   //    faSingleStepModeUnit22 : Bool;
   //    faSingleModeUnit22 : Bool;
   //    fctBit1ClampingUnit22 : Bool;
   //    fctBit2ClampingUnit22 : Bool;
   //    fctBit3ClampingUnit22 : Bool;
   //    prealarmOnUnit23 : Bool;
   //    messageOnUnit23 : Bool;
   //    faSetupModeUnit23 : Bool;
   //    faSingleStepModeUnit23 : Bool;
   //    faSingleModeUnit23 : Bool;
   //    fctBit1ClampingUnit23 : Bool;
   //    fctBit2ClampingUnit23 : Bool;
   //    fctBit3ClampingUnit23 : Bool;
   //    prealarmOnUnit24 : Bool;
   //    messageOnUnit24 : Bool;
   //    faSetupModeUnit24 : Bool;
   //    faSingleStepModeUnit24 : Bool;
   //    faSingleModeUnit24 : Bool;
   //    fctBit1ClampingUnit24 : Bool;
   //    fctBit2ClampingUnit24 : Bool;
   //    fctBit3ClampingUnit24 : Bool;
   //    prealarmOnUnit25 : Bool;
   //    messageOnUnit25 : Bool;
   //    faSetupModeUnit25 : Bool;
   //    faSingleStepModeUnit25 : Bool;
   //    faSingleModeUnit25 : Bool;
   //    fctBit1ClampingUnit25 : Bool;
   //    fctBit2ClampingUnit25 : Bool;
   //    fctBit3ClampingUnit25 : Bool;
   //    prealarmOnUnit26 : Bool;
   //    messageOnUnit26 : Bool;
   //    faSetupModeUnit26 : Bool;
   //    faSingleStepModeUnit26 : Bool;
   //    faSingleModeUnit26 : Bool;
   //    fctBit1ClampingUnit26 : Bool;
   //    fctBit2ClampingUnit26 : Bool;
   //    fctBit3ClampingUnit26 : Bool;
   //    prealarmOnUnit27 : Bool;
   //    messageOnUnit27 : Bool;
   //    faSetupModeUnit27 : Bool;
   //    faSingleStepModeUnit27 : Bool;
   //    faSingleModeUnit27 : Bool;
   //    fctBit1ClampingUnit27 : Bool;
   //    fctBit2ClampingUnit27 : Bool;
   //    fctBit3ClampingUnit27 : Bool;
   //    prealarmOnUnit28 : Bool;
   //    messageOnUnit28 : Bool;
   //    faSetupModeUnit28 : Bool;
   //    faSingleStepModeUnit28 : Bool;
   //    faSingleModeUnit28 : Bool;
   //    fctBit1ClampingUnit28 : Bool;
   //    fctBit2ClampingUnit28 : Bool;
   //    fctBit3ClampingUnit28 : Bool;
   //    prealarmOnUnit29 : Bool;
   //    messageOnUnit29 : Bool;
   //    faSetupModeUnit29 : Bool;
   //    faSingleStepModeUnit29 : Bool;
   //    faSingleModeUnit29 : Bool;
   //    fctBit1ClampingUnit29 : Bool;
   //    fctBit2ClampingUnit29 : Bool;
   //    fctBit3ClampingUnit29 : Bool;
   //    prealarmOnUnit30 : Bool;
   //    messageOnUnit30 : Bool;
   //    faSetupModeUnit30 : Bool;
   //    faSingleStepModeUnit30 : Bool;
   //    faSingleModeUnit30 : Bool;
   //    fctBit1ClampingUnit30 : Bool;
   //    fctBit2ClampingUnit30 : Bool;
   //    fctBit3ClampingUnit30 : Bool;
   //    prealarmOnUnit31 : Bool;
   //    messageOnUnit31 : Bool;
   //    faSetupModeUnit31 : Bool;
   //    faSingleStepModeUnit31 : Bool;
   //    faSingleModeUnit31 : Bool;
   //    fctBit1ClampingUnit31 : Bool;
   //    fctBit2ClampingUnit31 : Bool;
   //    fctBit3ClampingUnit31 : Bool;
   //    prealarmOnUnit32 : Bool;
   //    messageOnUnit32 : Bool;
   //    faSetupModeUnit32 : Bool;
   //    faSingleStepModeUnit32 : Bool;
   //    faSingleModeUnit32 : Bool;
   //    fctBit1ClampingUnit32 : Bool;
   //    fctBit2ClampingUnit32 : Bool;
   //    fctBit3ClampingUnit32 : Bool;
   //    prealarmOnUnit33 : Bool;
   //    messageOnUnit33 : Bool;
   //    faSetupModeUnit33 : Bool;
   //    faSingleStepModeUnit33 : Bool;
   //    faSingleModeUnit33 : Bool;
   //    fctBit1ClampingUnit33 : Bool;
   //    fctBit2ClampingUnit33 : Bool;
   //    fctBit3ClampingUnit33 : Bool;
   //    prealarmOnUnit34 : Bool;
   //    messageOnUnit34 : Bool;
   //    faSetupModeUnit34 : Bool;
   //    faSingleStepModeUnit34 : Bool;
   //    faSingleModeUnit34 : Bool;
   //    fctBit1ClampingUnit34 : Bool;
   //    fctBit2ClampingUnit34 : Bool;
   //    fctBit3ClampingUnit34 : Bool;
   //    prealarmOnUnit35 : Bool;
   //    messageOnUnit35 : Bool;
   //    faSetupModeUnit35 : Bool;
   //    faSingleStepModeUnit35 : Bool;
   //    faSingleModeUnit35 : Bool;
   //    fctBit1ClampingUnit35 : Bool;
   //    fctBit2ClampingUnit35 : Bool;
   //    fctBit3ClampingUnit35 : Bool;
   //    prealarmOnUnit36 : Bool;
   //    messageOnUnit36 : Bool;
   //    faSetupModeUnit36 : Bool;
   //    faSingleStepModeUnit36 : Bool;
   //    faSingleModeUnit36 : Bool;
   //    fctBit1ClampingUnit36 : Bool;
   //    fctBit2ClampingUnit36 : Bool;
   //    fctBit3ClampingUnit36 : Bool;
   //    prealarmOnUnit37 : Bool;
   //    messageOnUnit37 : Bool;
   //    faSetupModeUnit37 : Bool;
   //    faSingleStepModeUnit37 : Bool;
   //    faSingleModeUnit37 : Bool;
   //    fctBit1ClampingUnit37 : Bool;
   //    fctBit2ClampingUnit37 : Bool;
   //    fctBit3ClampingUnit37 : Bool;
   //    prealarmOnUnit38 : Bool;
   //    messageOnUnit38 : Bool;
   //    faSetupModeUnit38 : Bool;
   //    faSingleStepModeUnit38 : Bool;
   //    faSingleModeUnit38 : Bool;
   //    fctBit1ClampingUnit38 : Bool;
   //    fctBit2ClampingUnit38 : Bool;
   //    fctBit3ClampingUnit38 : Bool;
   //    prealarmOnUnit39 : Bool;
   //    messageOnUnit39 : Bool;
   //    faSetupModeUnit39 : Bool;
   //    faSingleStepModeUnit39 : Bool;
   //    faSingleModeUnit39 : Bool;
   //    fctBit1ClampingUnit39 : Bool;
   //    fctBit2ClampingUnit39 : Bool;
   //    fctBit3ClampingUnit39 : Bool;
   //    prealarmOnUnit40 : Bool;
   //    messageOnUnit40 : Bool;
   //    faSetupModeUnit40 : Bool;
   //    faSingleStepModeUnit40 : Bool;
   //    faSingleModeUnit40 : Bool;
   //    fctBit1ClampingUnit40 : Bool;
   //    fctBit2ClampingUnit40 : Bool;
   //    fctBit3ClampingUnit40 : Bool;
   //    targetCycleTimeCompleteMach : Word;
   //    targetCycleTime : Array[1..40] of Word;
   //    station : Array[1..40] of Word;
   //    directKeyScreen : Struct
   //       activeLine : Byte;
   //       singleMovementActive : Bool;
   //       singleLineSelected : Bool;
   //       singleLineRequestForLock : Bool;
   //       singleLineIsLockedByHMI : Bool;
   //       reserved2003p4 : Bool;
   //       reserved2003p5 : Bool;
   //       leftKeyPressedVDCK : Bool;
   //       rightKeyPressedVDCK : Bool;
   //    END_STRUCT;
   //    FC57_1 : DWord;
   //    FC57_2 : DWord;
   //    FC57_3 : Byte;
   //    FC57_4 : Byte;
   //    FC57_5 : Word;
   //    FC57_6 : Word;
   //    opKey2LeftVertical : Bool;
   //    opKey2RightVertical : Bool;
   //    opKey3LeftVertical : Bool;
   //    opKey3RightVertical : Bool;
   //    opKey4LeftVertical : Bool;
   //    opKey4RightVertical : Bool;
   //    opKey5LeftVertical : Bool;
   //    opKey5RightVertical : Bool;
   //    opKey6LeftVertical : Bool;
   //    opKey6RightVertical : Bool;
   //    opKey7LeftVertical : Bool;
   //    opKey7RightVertical : Bool;
   //    executionPlus : Bool;
   //    executionMinus : Bool;
   //    enableMotion : Bool;
   //    enablePCU : Bool;
   //    mppPlusKey : Bool;
   //    mppMinusKey : Bool;
   //    res2921 : Byte;
   //    typePreselectWorkpieceCode : Array[1..32] of Word;
   //    typePreselectColorChange : Array[1..32] of Bool;
   //    res2990 : Array[2990..2999] of Byte;
   //    unit1WorkpieceAMeas2 : Bool;
   //    unit1WorkpieceAMeas1 : Bool;
   //    unit1WorkpieceBMeas2 : Bool;
   //    unit1WorkpieceBMeas1 : Bool;
   //    unit1WorkpieceCMeas2 : Bool;
   //    unit1WorkpieceCMeas1 : Bool;
   //    unit1WorkpieceDMeas2 : Bool;
   //    unit1WorkpieceDMeas1 : Bool;
   //    unit1WorkpieceEMeas2 : Bool;
   //    unit1WorkpieceEMeas1 : Bool;
   //    unit1WorkpieceFMeas2 : Bool;
   //    unit1WorkpieceFMeas1 : Bool;
   //    unit1WorkpieceGMeas2 : Bool;
   //    unit1WorkpieceGMeas1 : Bool;
   //    unit1WorkpieceHMeas2 : Bool;
   //    unit1WorkpieceHMeas1 : Bool;
   //    unit2WorkpieceAMeas2 : Bool;
   //    unit2WorkpieceAMeas1 : Bool;
   //    unit2WorkpieceBMeas2 : Bool;
   //    unit2WorkpieceBMeas1 : Bool;
   //    unit2WorkpieceCMeas2 : Bool;
   //    unit2WorkpieceCMeas1 : Bool;
   //    unit2WorkpieceDMeas2 : Bool;
   //    unit2WorkpieceDMeas1 : Bool;
   //    unit2WorkpieceEMeas2 : Bool;
   //    unit2WorkpieceEMeas1 : Bool;
   //    unit2WorkpieceFMeas2 : Bool;
   //    unit2WorkpieceFMeas1 : Bool;
   //    unit2WorkpieceGMeas2 : Bool;
   //    unit2WorkpieceGMeas1 : Bool;
   //    unit2WorkpieceHMeas2 : Bool;
   //    unit2WorkpieceHMeas1 : Bool;
   //    unit3WorkpieceAMeas2 : Bool;
   //    unit3WorkpieceAMeas1 : Bool;
   //    unit3WorkpieceBMeas2 : Bool;
   //    unit3WorkpieceBMeas1 : Bool;
   //    unit3WorkpieceCMeas2 : Bool;
   //    unit3WorkpieceCMeas1 : Bool;
   //    unit3WorkpieceDMeas2 : Bool;
   //    unit3WorkpieceDMeas1 : Bool;
   //    unit3WorkpieceEMeas2 : Bool;
   //    unit3WorkpieceEMeas1 : Bool;
   //    unit3WorkpieceFMeas2 : Bool;
   //    unit3WorkpieceFMeas1 : Bool;
   //    unit3WorkpieceGMeas2 : Bool;
   //    unit3WorkpieceGMeas1 : Bool;
   //    unit3WorkpieceHMeas2 : Bool;
   //    unit3WorkpieceHMeas1 : Bool;
   //    unit4WorkpieceAMeas2 : Bool;
   //    unit4WorkpieceAMeas1 : Bool;
   //    unit4WorkpieceBMeas2 : Bool;
   //    unit4WorkpieceBMeas1 : Bool;
   //    unit4WorkpieceCMeas2 : Bool;
   //    unit4WorkpieceCMeas1 : Bool;
   //    unit4WorkpieceDMeas2 : Bool;
   //    unit4WorkpieceDMeas1 : Bool;
   //    unit4WorkpieceEMeas2 : Bool;
   //    unit4WorkpieceEMeas1 : Bool;
   //    unit4WorkpieceFMeas2 : Bool;
   //    unit4WorkpieceFMeas1 : Bool;
   //    unit4WorkpieceGMeas2 : Bool;
   //    unit4WorkpieceGMeas1 : Bool;
   //    unit4WorkpieceHMeas2 : Bool;
   //    unit4WorkpieceHMeas1 : Bool;
   //    unit5WorkpieceAMeas2 : Bool;
   //    unit5WorkpieceAMeas1 : Bool;
   //    unit5WorkpieceBMeas2 : Bool;
   //    unit5WorkpieceBMeas1 : Bool;
   //    unit5WorkpieceCMeas2 : Bool;
   //    unit5WorkpieceCMeas1 : Bool;
   //    unit5WorkpieceDMeas2 : Bool;
   //    unit5WorkpieceDMeas1 : Bool;
   //    unit5WorkpieceEMeas2 : Bool;
   //    unit5WorkpieceEMeas1 : Bool;
   //    unit5WorkpieceFMeas2 : Bool;
   //    unit5WorkpieceFMeas1 : Bool;
   //    unit5WorkpieceGMeas2 : Bool;
   //    unit5WorkpieceGMeas1 : Bool;
   //    unit5WorkpieceHMeas2 : Bool;
   //    unit5WorkpieceHMeas1 : Bool;
   //    unit6WorkpieceAMeas2 : Bool;
   //    unit6WorkpieceAMeas1 : Bool;
   //    unit6WorkpieceBMeas2 : Bool;
   //    unit6WorkpieceBMeas1 : Bool;
   //    unit6WorkpieceCMeas2 : Bool;
   //    unit6WorkpieceCMeas1 : Bool;
   //    unit6WorkpieceDMeas2 : Bool;
   //    unit6WorkpieceDMeas1 : Bool;
   //    unit6WorkpieceEMeas2 : Bool;
   //    unit6WorkpieceEMeas1 : Bool;
   //    unit6WorkpieceFMeas2 : Bool;
   //    unit6WorkpieceFMeas1 : Bool;
   //    unit6WorkpieceGMeas2 : Bool;
   //    unit6WorkpieceGMeas1 : Bool;
   //    unit6WorkpieceHMeas2 : Bool;
   //    unit6WorkpieceHMeas1 : Bool;
   //    unit7WorkpieceAMeas2 : Bool;
   //    unit7WorkpieceAMeas1 : Bool;
   //    unit7WorkpieceBMeas2 : Bool;
   //    unit7WorkpieceBMeas1 : Bool;
   //    unit7WorkpieceCMeas2 : Bool;
   //    unit7WorkpieceCMeas1 : Bool;
   //    unit7WorkpieceDMeas2 : Bool;
   //    unit7WorkpieceDMeas1 : Bool;
   //    unit7WorkpieceEMeas2 : Bool;
   //    unit7WorkpieceEMeas1 : Bool;
   //    unit7WorkpieceFMeas2 : Bool;
   //    unit7WorkpieceFMeas1 : Bool;
   //    unit7WorkpieceGMeas2 : Bool;
   //    unit7WorkpieceGMeas1 : Bool;
   //    unit7WorkpieceHMeas2 : Bool;
   //    unit7WorkpieceHMeas1 : Bool;
   //    unit8WorkpieceAMeas2 : Bool;
   //    unit8WorkpieceAMeas1 : Bool;
   //    unit8WorkpieceBMeas2 : Bool;
   //    unit8WorkpieceBMeas1 : Bool;
   //    unit8WorkpieceCMeas2 : Bool;
   //    unit8WorkpieceCMeas1 : Bool;
   //    unit8WorkpieceDMeas2 : Bool;
   //    unit8WorkpieceDMeas1 : Bool;
   //    unit8WorkpieceEMeas2 : Bool;
   //    unit8WorkpieceEMeas1 : Bool;
   //    unit8WorkpieceFMeas2 : Bool;
   //    unit8WorkpieceFMeas1 : Bool;
   //    unit8WorkpieceGMeas2 : Bool;
   //    unit8WorkpieceGMeas1 : Bool;
   //    unit8WorkpieceHMeas2 : Bool;
   //    unit8WorkpieceHMeas1 : Bool;
   //    unit9WorkpieceAMeas2 : Bool;
   //    unit9WorkpieceAMeas1 : Bool;
   //    unit9WorkpieceBMeas2 : Bool;
   //    unit9WorkpieceBMeas1 : Bool;
   //    unit9WorkpieceCMeas2 : Bool;
   //    unit9WorkpieceCMeas1 : Bool;
   //    unit9WorkpieceDMeas2 : Bool;
   //    unit9WorkpieceDMeas1 : Bool;
   //    unit9WorkpieceEMeas2 : Bool;
   //    unit9WorkpieceEMeas1 : Bool;
   //    unit9WorkpieceFMeas2 : Bool;
   //    unit9WorkpieceFMeas1 : Bool;
   //    unit9WorkpieceGMeas2 : Bool;
   //    unit9WorkpieceGMeas1 : Bool;
   //    unit9WorkpieceHMeas2 : Bool;
   //    unit9WorkpieceHMeas1 : Bool;
   //    unit10WorkpieceAMeas2 : Bool;
   //    unit10WorkpieceAMeas1 : Bool;
   //    unit10WorkpieceBMeas2 : Bool;
   //    unit10WorkpieceBMeas1 : Bool;
   //    unit10WorkpieceCMeas2 : Bool;
   //    unit10WorkpieceCMeas1 : Bool;
   //    unit10WorkpieceDMeas2 : Bool;
   //    unit10WorkpieceDMeas1 : Bool;
   //    unit10WorkpieceEMeas2 : Bool;
   //    unit10WorkpieceEMeas1 : Bool;
   //    unit10WorkpieceFMeas2 : Bool;
   //    unit10WorkpieceFMeas1 : Bool;
   //    unit10WorkpieceGMeas2 : Bool;
   //    unit10WorkpieceGMeas1 : Bool;
   //    unit10WorkpieceHMeas2 : Bool;
   //    unit10WorkpieceHMeas1 : Bool;
   //    unit11WorkpieceAMeas2 : Bool;
   //    unit11WorkpieceAMeas1 : Bool;
   //    unit11WorkpieceBMeas2 : Bool;
   //    unit11WorkpieceBMeas1 : Bool;
   //    unit11WorkpieceCMeas2 : Bool;
   //    unit11WorkpieceCMeas1 : Bool;
   //    unit11WorkpieceDMeas2 : Bool;
   //    unit11WorkpieceDMeas1 : Bool;
   //    unit11WorkpieceEMeas2 : Bool;
   //    unit11WorkpieceEMeas1 : Bool;
   //    unit11WorkpieceFMeas2 : Bool;
   //    unit11WorkpieceFMeas1 : Bool;
   //    unit11WorkpieceGMeas2 : Bool;
   //    unit11WorkpieceGMeas1 : Bool;
   //    unit11WorkpieceHMeas2 : Bool;
   //    unit11WorkpieceHMeas1 : Bool;
   //    unit12WorkpieceAMeas2 : Bool;
   //    unit12WorkpieceAMeas1 : Bool;
   //    unit12WorkpieceBMeas2 : Bool;
   //    unit12WorkpieceBMeas1 : Bool;
   //    unit12WorkpieceCMeas2 : Bool;
   //    unit12WorkpieceCMeas1 : Bool;
   //    unit12WorkpieceDMeas2 : Bool;
   //    unit12WorkpieceDMeas1 : Bool;
   //    unit12WorkpieceEMeas2 : Bool;
   //    unit12WorkpieceEMeas1 : Bool;
   //    unit12WorkpieceFMeas2 : Bool;
   //    unit12WorkpieceFMeas1 : Bool;
   //    unit12WorkpieceGMeas2 : Bool;
   //    unit12WorkpieceGMeas1 : Bool;
   //    unit12WorkpieceHMeas2 : Bool;
   //    unit12WorkpieceHMeas1 : Bool;
   //    unit13WorkpieceAMeas2 : Bool;
   //    unit13WorkpieceAMeas1 : Bool;
   //    unit13WorkpieceBMeas2 : Bool;
   //    unit13WorkpieceBMeas1 : Bool;
   //    unit13WorkpieceCMeas2 : Bool;
   //    unit13WorkpieceCMeas1 : Bool;
   //    unit13WorkpieceDMeas2 : Bool;
   //    unit13WorkpieceDMeas1 : Bool;
   //    unit13WorkpieceEMeas2 : Bool;
   //    unit13WorkpieceEMeas1 : Bool;
   //    unit13WorkpieceFMeas2 : Bool;
   //    unit13WorkpieceFMeas1 : Bool;
   //    unit13WorkpieceGMeas2 : Bool;
   //    unit13WorkpieceGMeas1 : Bool;
   //    unit13WorkpieceHMeas2 : Bool;
   //    unit13WorkpieceHMeas1 : Bool;
   //    unit14WorkpieceAMeas2 : Bool;
   //    unit14WorkpieceAMeas1 : Bool;
   //    unit14WorkpieceBMeas2 : Bool;
   //    unit14WorkpieceBMeas1 : Bool;
   //    unit14WorkpieceCMeas2 : Bool;
   //    unit14WorkpieceCMeas1 : Bool;
   //    unit14WorkpieceDMeas2 : Bool;
   //    unit14WorkpieceDMeas1 : Bool;
   //    unit14WorkpieceEMeas2 : Bool;
   //    unit14WorkpieceEMeas1 : Bool;
   //    unit14WorkpieceFMeas2 : Bool;
   //    unit14WorkpieceFMeas1 : Bool;
   //    unit14WorkpieceGMeas2 : Bool;
   //    unit14WorkpieceGMeas1 : Bool;
   //    unit14WorkpieceHMeas2 : Bool;
   //    unit14WorkpieceHMeas1 : Bool;
   //    unit15WorkpieceAMeas2 : Bool;
   //    unit15WorkpieceAMeas1 : Bool;
   //    unit15WorkpieceBMeas2 : Bool;
   //    unit15WorkpieceBMeas1 : Bool;
   //    unit15WorkpieceCMeas2 : Bool;
   //    unit15WorkpieceCMeas1 : Bool;
   //    unit15WorkpieceDMeas2 : Bool;
   //    unit15WorkpieceDMeas1 : Bool;
   //    unit15WorkpieceEMeas2 : Bool;
   //    unit15WorkpieceEMeas1 : Bool;
   //    unit15WorkpieceFMeas2 : Bool;
   //    unit15WorkpieceFMeas1 : Bool;
   //    unit15WorkpieceGMeas2 : Bool;
   //    unit15WorkpieceGMeas1 : Bool;
   //    unit15WorkpieceHMeas2 : Bool;
   //    unit15WorkpieceHMeas1 : Bool;
   //    unit16WorkpieceAMeas2 : Bool;
   //    unit16WorkpieceAMeas1 : Bool;
   //    unit16WorkpieceBMeas2 : Bool;
   //    unit16WorkpieceBMeas1 : Bool;
   //    unit16WorkpieceCMeas2 : Bool;
   //    unit16WorkpieceCMeas1 : Bool;
   //    unit16WorkpieceDMeas2 : Bool;
   //    unit16WorkpieceDMeas1 : Bool;
   //    unit16WorkpieceEMeas2 : Bool;
   //    unit16WorkpieceEMeas1 : Bool;
   //    unit16WorkpieceFMeas2 : Bool;
   //    unit16WorkpieceFMeas1 : Bool;
   //    unit16WorkpieceGMeas2 : Bool;
   //    unit16WorkpieceGMeas1 : Bool;
   //    unit16WorkpieceHMeas2 : Bool;
   //    unit16WorkpieceHMeas1 : Bool;
   //    unit17WorkpieceAMeas2 : Bool;
   //    unit17WorkpieceAMeas1 : Bool;
   //    unit17WorkpieceBMeas2 : Bool;
   //    unit17WorkpieceBMeas1 : Bool;
   //    unit17WorkpieceCMeas2 : Bool;
   //    unit17WorkpieceCMeas1 : Bool;
   //    unit17WorkpieceDMeas2 : Bool;
   //    unit17WorkpieceDMeas1 : Bool;
   //    unit17WorkpieceEMeas2 : Bool;
   //    unit17WorkpieceEMeas1 : Bool;
   //    unit17WorkpieceFMeas2 : Bool;
   //    unit17WorkpieceFMeas1 : Bool;
   //    unit17WorkpieceGMeas2 : Bool;
   //    unit17WorkpieceGMeas1 : Bool;
   //    unit17WorkpieceHMeas2 : Bool;
   //    unit17WorkpieceHMeas1 : Bool;
   //    unit18WorkpieceAMeas2 : Bool;
   //    unit18WorkpieceAMeas1 : Bool;
   //    unit18WorkpieceBMeas2 : Bool;
   //    unit18WorkpieceBMeas1 : Bool;
   //    unit18WorkpieceCMeas2 : Bool;
   //    unit18WorkpieceCMeas1 : Bool;
   //    unit18WorkpieceDMeas2 : Bool;
   //    unit18WorkpieceDMeas1 : Bool;
   //    unit18WorkpieceEMeas2 : Bool;
   //    unit18WorkpieceEMeas1 : Bool;
   //    unit18WorkpieceFMeas2 : Bool;
   //    unit18WorkpieceFMeas1 : Bool;
   //    unit18WorkpieceGMeas2 : Bool;
   //    unit18WorkpieceGMeas1 : Bool;
   //    unit18WorkpieceHMeas2 : Bool;
   //    unit18WorkpieceHMeas1 : Bool;
   //    unit19WorkpieceAMeas2 : Bool;
   //    unit19WorkpieceAMeas1 : Bool;
   //    unit19WorkpieceBMeas2 : Bool;
   //    unit19WorkpieceBMeas1 : Bool;
   //    unit19WorkpieceCMeas2 : Bool;
   //    unit19WorkpieceCMeas1 : Bool;
   //    unit19WorkpieceDMeas2 : Bool;
   //    unit19WorkpieceDMeas1 : Bool;
   //    unit19WorkpieceEMeas2 : Bool;
   //    unit19WorkpieceEMeas1 : Bool;
   //    unit19WorkpieceFMeas2 : Bool;
   //    unit19WorkpieceFMeas1 : Bool;
   //    unit19WorkpieceGMeas2 : Bool;
   //    unit19WorkpieceGMeas1 : Bool;
   //    unit19WorkpieceHMeas2 : Bool;
   //    unit19WorkpieceHMeas1 : Bool;
   //    unit20WorkpieceAMeas2 : Bool;
   //    unit20WorkpieceAMeas1 : Bool;
   //    unit20WorkpieceBMeas2 : Bool;
   //    unit20WorkpieceBMeas1 : Bool;
   //    unit20WorkpieceCMeas2 : Bool;
   //    unit20WorkpieceCMeas1 : Bool;
   //    unit20WorkpieceDMeas2 : Bool;
   //    unit20WorkpieceDMeas1 : Bool;
   //    unit20WorkpieceEMeas2 : Bool;
   //    unit20WorkpieceEMeas1 : Bool;
   //    unit20WorkpieceFMeas2 : Bool;
   //    unit20WorkpieceFMeas1 : Bool;
   //    unit20WorkpieceGMeas2 : Bool;
   //    unit20WorkpieceGMeas1 : Bool;
   //    unit20WorkpieceHMeas2 : Bool;
   //    unit20WorkpieceHMeas1 : Bool;
   //    unit21WorkpieceAMeas2 : Bool;
   //    unit21WorkpieceAMeas1 : Bool;
   //    unit21WorkpieceBMeas2 : Bool;
   //    unit21WorkpieceBMeas1 : Bool;
   //    unit21WorkpieceCMeas2 : Bool;
   //    unit21WorkpieceCMeas1 : Bool;
   //    unit21WorkpieceDMeas2 : Bool;
   //    unit21WorkpieceDMeas1 : Bool;
   //    unit21WorkpieceEMeas2 : Bool;
   //    unit21WorkpieceEMeas1 : Bool;
   //    unit21WorkpieceFMeas2 : Bool;
   //    unit21WorkpieceFMeas1 : Bool;
   //    unit21WorkpieceGMeas2 : Bool;
   //    unit21WorkpieceGMeas1 : Bool;
   //    unit21WorkpieceHMeas2 : Bool;
   //    unit21WorkpieceHMeas1 : Bool;
   //    unit22WorkpieceAMeas2 : Bool;
   //    unit22WorkpieceAMeas1 : Bool;
   //    unit22WorkpieceBMeas2 : Bool;
   //    unit22WorkpieceBMeas1 : Bool;
   //    unit22WorkpieceCMeas2 : Bool;
   //    unit22WorkpieceCMeas1 : Bool;
   //    unit22WorkpieceDMeas2 : Bool;
   //    unit22WorkpieceDMeas1 : Bool;
   //    unit22WorkpieceEMeas2 : Bool;
   //    unit22WorkpieceEMeas1 : Bool;
   //    unit22WorkpieceFMeas2 : Bool;
   //    unit22WorkpieceFMeas1 : Bool;
   //    unit22WorkpieceGMeas2 : Bool;
   //    unit22WorkpieceGMeas1 : Bool;
   //    unit22WorkpieceHMeas2 : Bool;
   //    unit22WorkpieceHMeas1 : Bool;
   //    unit23WorkpieceAMeas2 : Bool;
   //    unit23WorkpieceAMeas1 : Bool;
   //    unit23WorkpieceBMeas2 : Bool;
   //    unit23WorkpieceBMeas1 : Bool;
   //    unit23WorkpieceCMeas2 : Bool;
   //    unit23WorkpieceCMeas1 : Bool;
   //    unit23WorkpieceDMeas2 : Bool;
   //    unit23WorkpieceDMeas1 : Bool;
   //    unit23WorkpieceEMeas2 : Bool;
   //    unit23WorkpieceEMeas1 : Bool;
   //    unit23WorkpieceFMeas2 : Bool;
   //    unit23WorkpieceFMeas1 : Bool;
   //    unit23WorkpieceGMeas2 : Bool;
   //    unit23WorkpieceGMeas1 : Bool;
   //    unit23WorkpieceHMeas2 : Bool;
   //    unit23WorkpieceHMeas1 : Bool;
   //    unit24WorkpieceAMeas2 : Bool;
   //    unit24WorkpieceAMeas1 : Bool;
   //    unit24WorkpieceBMeas2 : Bool;
   //    unit24WorkpieceBMeas1 : Bool;
   //    unit24WorkpieceCMeas2 : Bool;
   //    unit24WorkpieceCMeas1 : Bool;
   //    unit24WorkpieceDMeas2 : Bool;
   //    unit24WorkpieceDMeas1 : Bool;
   //    unit24WorkpieceEMeas2 : Bool;
   //    unit24WorkpieceEMeas1 : Bool;
   //    unit24WorkpieceFMeas2 : Bool;
   //    unit24WorkpieceFMeas1 : Bool;
   //    unit24WorkpieceGMeas2 : Bool;
   //    unit24WorkpieceGMeas1 : Bool;
   //    unit24WorkpieceHMeas2 : Bool;
   //    unit24WorkpieceHMeas1 : Bool;
   //    unit25WorkpieceAMeas2 : Bool;
   //    unit25WorkpieceAMeas1 : Bool;
   //    unit25WorkpieceBMeas2 : Bool;
   //    unit25WorkpieceBMeas1 : Bool;
   //    unit25WorkpieceCMeas2 : Bool;
   //    unit25WorkpieceCMeas1 : Bool;
   //    unit25WorkpieceDMeas2 : Bool;
   //    unit25WorkpieceDMeas1 : Bool;
   //    unit25WorkpieceEMeas2 : Bool;
   //    unit25WorkpieceEMeas1 : Bool;
   //    unit25WorkpieceFMeas2 : Bool;
   //    unit25WorkpieceFMeas1 : Bool;
   //    unit25WorkpieceGMeas2 : Bool;
   //    unit25WorkpieceGMeas1 : Bool;
   //    unit25WorkpieceHMeas2 : Bool;
   //    unit25WorkpieceHMeas1 : Bool;
   //    unit26WorkpieceAMeas2 : Bool;
   //    unit26WorkpieceAMeas1 : Bool;
   //    unit26WorkpieceBMeas2 : Bool;
   //    unit26WorkpieceBMeas1 : Bool;
   //    unit26WorkpieceCMeas2 : Bool;
   //    unit26WorkpieceCMeas1 : Bool;
   //    unit26WorkpieceDMeas2 : Bool;
   //    unit26WorkpieceDMeas1 : Bool;
   //    unit26WorkpieceEMeas2 : Bool;
   //    unit26WorkpieceEMeas1 : Bool;
   //    unit26WorkpieceFMeas2 : Bool;
   //    unit26WorkpieceFMeas1 : Bool;
   //    unit26WorkpieceGMeas2 : Bool;
   //    unit26WorkpieceGMeas1 : Bool;
   //    unit26WorkpieceHMeas2 : Bool;
   //    unit26WorkpieceHMeas1 : Bool;
   //    unit27WorkpieceAMeas2 : Bool;
   //    unit27WorkpieceAMeas1 : Bool;
   //    unit27WorkpieceBMeas2 : Bool;
   //    unit27WorkpieceBMeas1 : Bool;
   //    unit27WorkpieceCMeas2 : Bool;
   //    unit27WorkpieceCMeas1 : Bool;
   //    unit27WorkpieceDMeas2 : Bool;
   //    unit27WorkpieceDMeas1 : Bool;
   //    unit27WorkpieceEMeas2 : Bool;
   //    unit27WorkpieceEMeas1 : Bool;
   //    unit27WorkpieceFMeas2 : Bool;
   //    unit27WorkpieceFMeas1 : Bool;
   //    unit27WorkpieceGMeas2 : Bool;
   //    unit27WorkpieceGMeas1 : Bool;
   //    unit27WorkpieceHMeas2 : Bool;
   //    unit27WorkpieceHMeas1 : Bool;
   //    unit28WorkpieceAMeas2 : Bool;
   //    unit28WorkpieceAMeas1 : Bool;
   //    unit28WorkpieceBMeas2 : Bool;
   //    unit28WorkpieceBMeas1 : Bool;
   //    unit28WorkpieceCMeas2 : Bool;
   //    unit28WorkpieceCMeas1 : Bool;
   //    unit28WorkpieceDMeas2 : Bool;
   //    unit28WorkpieceDMeas1 : Bool;
   //    unit28WorkpieceEMeas2 : Bool;
   //    unit28WorkpieceEMeas1 : Bool;
   //    unit28WorkpieceFMeas2 : Bool;
   //    unit28WorkpieceFMeas1 : Bool;
   //    unit28WorkpieceGMeas2 : Bool;
   //    unit28WorkpieceGMeas1 : Bool;
   //    unit28WorkpieceHMeas2 : Bool;
   //    unit28WorkpieceHMeas1 : Bool;
   //    unit29WorkpieceAMeas2 : Bool;
   //    unit29WorkpieceAMeas1 : Bool;
   //    unit29WorkpieceBMeas2 : Bool;
   //    unit29WorkpieceBMeas1 : Bool;
   //    unit29WorkpieceCMeas2 : Bool;
   //    unit29WorkpieceCMeas1 : Bool;
   //    unit29WorkpieceDMeas2 : Bool;
   //    unit29WorkpieceDMeas1 : Bool;
   //    unit29WorkpieceEMeas2 : Bool;
   //    unit29WorkpieceEMeas1 : Bool;
   //    unit29WorkpieceFMeas2 : Bool;
   //    unit29WorkpieceFMeas1 : Bool;
   //    unit29WorkpieceGMeas2 : Bool;
   //    unit29WorkpieceGMeas1 : Bool;
   //    unit29WorkpieceHMeas2 : Bool;
   //    unit29WorkpieceHMeas1 : Bool;
   //    unit30WorkpieceAMeas2 : Bool;
   //    unit30WorkpieceAMeas1 : Bool;
   //    unit30WorkpieceBMeas2 : Bool;
   //    unit30WorkpieceBMeas1 : Bool;
   //    unit30WorkpieceCMeas2 : Bool;
   //    unit30WorkpieceCMeas1 : Bool;
   //    unit30WorkpieceDMeas2 : Bool;
   //    unit30WorkpieceDMeas1 : Bool;
   //    unit30WorkpieceEMeas2 : Bool;
   //    unit30WorkpieceEMeas1 : Bool;
   //    unit30WorkpieceFMeas2 : Bool;
   //    unit30WorkpieceFMeas1 : Bool;
   //    unit30WorkpieceGMeas2 : Bool;
   //    unit30WorkpieceGMeas1 : Bool;
   //    unit30WorkpieceHMeas2 : Bool;
   //    unit30WorkpieceHMeas1 : Bool;
   //    unit31WorkpieceAMeas2 : Bool;
   //    unit31WorkpieceAMeas1 : Bool;
   //    unit31WorkpieceBMeas2 : Bool;
   //    unit31WorkpieceBMeas1 : Bool;
   //    unit31WorkpieceCMeas2 : Bool;
   //    unit31WorkpieceCMeas1 : Bool;
   //    unit31WorkpieceDMeas2 : Bool;
   //    unit31WorkpieceDMeas1 : Bool;
   //    unit31WorkpieceEMeas2 : Bool;
   //    unit31WorkpieceEMeas1 : Bool;
   //    unit31WorkpieceFMeas2 : Bool;
   //    unit31WorkpieceFMeas1 : Bool;
   //    unit31WorkpieceGMeas2 : Bool;
   //    unit31WorkpieceGMeas1 : Bool;
   //    unit31WorkpieceHMeas2 : Bool;
   //    unit31WorkpieceHMeas1 : Bool;
   //    unit32WorkpieceAMeas2 : Bool;
   //    unit32WorkpieceAMeas1 : Bool;
   //    unit32WorkpieceBMeas2 : Bool;
   //    unit32WorkpieceBMeas1 : Bool;
   //    unit32WorkpieceCMeas2 : Bool;
   //    unit32WorkpieceCMeas1 : Bool;
   //    unit32WorkpieceDMeas2 : Bool;
   //    unit32WorkpieceDMeas1 : Bool;
   //    unit32WorkpieceEMeas2 : Bool;
   //    unit32WorkpieceEMeas1 : Bool;
   //    unit32WorkpieceFMeas2 : Bool;
   //    unit32WorkpieceFMeas1 : Bool;
   //    unit32WorkpieceGMeas2 : Bool;
   //    unit32WorkpieceGMeas1 : Bool;
   //    unit32WorkpieceHMeas2 : Bool;
   //    unit32WorkpieceHMeas1 : Bool;
   //    unit33WorkpieceAMeas2 : Bool;
   //    unit33WorkpieceAMeas1 : Bool;
   //    unit33WorkpieceBMeas2 : Bool;
   //    unit33WorkpieceBMeas1 : Bool;
   //    unit33WorkpieceCMeas2 : Bool;
   //    unit33WorkpieceCMeas1 : Bool;
   //    unit33WorkpieceDMeas2 : Bool;
   //    unit33WorkpieceDMeas1 : Bool;
   //    unit33WorkpieceEMeas2 : Bool;
   //    unit33WorkpieceEMeas1 : Bool;
   //    unit33WorkpieceFMeas2 : Bool;
   //    unit33WorkpieceFMeas1 : Bool;
   //    unit33WorkpieceGMeas2 : Bool;
   //    unit33WorkpieceGMeas1 : Bool;
   //    unit33WorkpieceHMeas2 : Bool;
   //    unit33WorkpieceHMeas1 : Bool;
   //    unit34WorkpieceAMeas2 : Bool;
   //    unit34WorkpieceAMeas1 : Bool;
   //    unit34WorkpieceBMeas2 : Bool;
   //    unit34WorkpieceBMeas1 : Bool;
   //    unit34WorkpieceCMeas2 : Bool;
   //    unit34WorkpieceCMeas1 : Bool;
   //    unit34WorkpieceDMeas2 : Bool;
   //    unit34WorkpieceDMeas1 : Bool;
   //    unit34WorkpieceEMeas2 : Bool;
   //    unit34WorkpieceEMeas1 : Bool;
   //    unit34WorkpieceFMeas2 : Bool;
   //    unit34WorkpieceFMeas1 : Bool;
   //    unit34WorkpieceGMeas2 : Bool;
   //    unit34WorkpieceGMeas1 : Bool;
   //    unit34WorkpieceHMeas2 : Bool;
   //    unit34WorkpieceHMeas1 : Bool;
   //    unit35WorkpieceAMeas2 : Bool;
   //    unit35WorkpieceAMeas1 : Bool;
   //    unit35WorkpieceBMeas2 : Bool;
   //    unit35WorkpieceBMeas1 : Bool;
   //    unit35WorkpieceCMeas2 : Bool;
   //    unit35WorkpieceCMeas1 : Bool;
   //    unit35WorkpieceDMeas2 : Bool;
   //    unit35WorkpieceDMeas1 : Bool;
   //    unit35WorkpieceEMeas2 : Bool;
   //    unit35WorkpieceEMeas1 : Bool;
   //    unit35WorkpieceFMeas2 : Bool;
   //    unit35WorkpieceFMeas1 : Bool;
   //    unit35WorkpieceGMeas2 : Bool;
   //    unit35WorkpieceGMeas1 : Bool;
   //    unit35WorkpieceHMeas2 : Bool;
   //    unit35WorkpieceHMeas1 : Bool;
   //    unit36WorkpieceAMeas2 : Bool;
   //    unit36WorkpieceAMeas1 : Bool;
   //    unit36WorkpieceBMeas2 : Bool;
   //    unit36WorkpieceBMeas1 : Bool;
   //    unit36WorkpieceCMeas2 : Bool;
   //    unit36WorkpieceCMeas1 : Bool;
   //    unit36WorkpieceDMeas2 : Bool;
   //    unit36WorkpieceDMeas1 : Bool;
   //    unit36WorkpieceEMeas2 : Bool;
   //    unit36WorkpieceEMeas1 : Bool;
   //    unit36WorkpieceFMeas2 : Bool;
   //    unit36WorkpieceFMeas1 : Bool;
   //    unit36WorkpieceGMeas2 : Bool;
   //    unit36WorkpieceGMeas1 : Bool;
   //    unit36WorkpieceHMeas2 : Bool;
   //    unit36WorkpieceHMeas1 : Bool;
   //    unit37WorkpieceAMeas2 : Bool;
   //    unit37WorkpieceAMeas1 : Bool;
   //    unit37WorkpieceBMeas2 : Bool;
   //    unit37WorkpieceBMeas1 : Bool;
   //    unit37WorkpieceCMeas2 : Bool;
   //    unit37WorkpieceCMeas1 : Bool;
   //    unit37WorkpieceDMeas2 : Bool;
   //    unit37WorkpieceDMeas1 : Bool;
   //    unit37WorkpieceEMeas2 : Bool;
   //    unit37WorkpieceEMeas1 : Bool;
   //    unit37WorkpieceFMeas2 : Bool;
   //    unit37WorkpieceFMeas1 : Bool;
   //    unit37WorkpieceGMeas2 : Bool;
   //    unit37WorkpieceGMeas1 : Bool;
   //    unit37WorkpieceHMeas2 : Bool;
   //    unit37WorkpieceHMeas1 : Bool;
   //    unit38WorkpieceAMeas2 : Bool;
   //    unit38WorkpieceAMeas1 : Bool;
   //    unit38WorkpieceBMeas2 : Bool;
   //    unit38WorkpieceBMeas1 : Bool;
   //    unit38WorkpieceCMeas2 : Bool;
   //    unit38WorkpieceCMeas1 : Bool;
   //    unit38WorkpieceDMeas2 : Bool;
   //    unit38WorkpieceDMeas1 : Bool;
   //    unit38WorkpieceEMeas2 : Bool;
   //    unit38WorkpieceEMeas1 : Bool;
   //    unit38WorkpieceFMeas2 : Bool;
   //    unit38WorkpieceFMeas1 : Bool;
   //    unit38WorkpieceGMeas2 : Bool;
   //    unit38WorkpieceGMeas1 : Bool;
   //    unit38WorkpieceHMeas2 : Bool;
   //    unit38WorkpieceHMeas1 : Bool;
   //    unit39WorkpieceAMeas2 : Bool;
   //    unit39WorkpieceAMeas1 : Bool;
   //    unit39WorkpieceBMeas2 : Bool;
   //    unit39WorkpieceBMeas1 : Bool;
   //    unit39WorkpieceCMeas2 : Bool;
   //    unit39WorkpieceCMeas1 : Bool;
   //    unit39WorkpieceDMeas2 : Bool;
   //    unit39WorkpieceDMeas1 : Bool;
   //    unit39WorkpieceEMeas2 : Bool;
   //    unit39WorkpieceEMeas1 : Bool;
   //    unit39WorkpieceFMeas2 : Bool;
   //    unit39WorkpieceFMeas1 : Bool;
   //    unit39WorkpieceGMeas2 : Bool;
   //    unit39WorkpieceGMeas1 : Bool;
   //    unit39WorkpieceHMeas2 : Bool;
   //    unit39WorkpieceHMeas1 : Bool;
   //    unit40WorkpieceAMeas2 : Bool;
   //    unit40WorkpieceAMeas1 : Bool;
   //    unit40WorkpieceBMeas2 : Bool;
   //    unit40WorkpieceBMeas1 : Bool;
   //    unit40WorkpieceCMeas2 : Bool;
   //    unit40WorkpieceCMeas1 : Bool;
   //    unit40WorkpieceDMeas2 : Bool;
   //    unit40WorkpieceDMeas1 : Bool;
   //    unit40WorkpieceEMeas2 : Bool;
   //    unit40WorkpieceEMeas1 : Bool;
   //    unit40WorkpieceFMeas2 : Bool;
   //    unit40WorkpieceFMeas1 : Bool;
   //    unit40WorkpieceGMeas2 : Bool;
   //    unit40WorkpieceGMeas1 : Bool;
   //    unit40WorkpieceHMeas2 : Bool;
   //    unit40WorkpieceHMeas1 : Bool;
   //    workpieceStatusUnit01_01 : Bool;
   //    workpieceStatusUnit01_11 : Bool;
   //    workpieceStatusUnit02_01 : Bool;
   //    workpieceStatusUnit02_11 : Bool;
   //    workpieceStatusUnit03_01 : Bool;
   //    workpieceStatusUnit03_11 : Bool;
   //    workpieceStatusUnit04_01 : Bool;
   //    workpieceStatusUnit04_11 : Bool;
   //    workpieceStatusUnit05_01 : Bool;
   //    workpieceStatusUnit05_11 : Bool;
   //    workpieceStatusUnit06_01 : Bool;
   //    workpieceStatusUnit06_11 : Bool;
   //    workpieceStatusUnit07_01 : Bool;
   //    workpieceStatusUnit07_11 : Bool;
   //    workpieceStatusUnit08_01 : Bool;
   //    workpieceStatusUnit08_11 : Bool;
   //    workpieceStatusUnit09_01 : Bool;
   //    workpieceStatusUnit09_11 : Bool;
   //    workpieceStatusUnit10_01 : Bool;
   //    workpieceStatusUnit10_11 : Bool;
   //    workpieceStatusUnit11_01 : Bool;
   //    workpieceStatusUnit11_11 : Bool;
   //    workpieceStatusUnit12_01 : Bool;
   //    workpieceStatusUnit12_11 : Bool;
   //    workpieceStatusUnit13_01 : Bool;
   //    workpieceStatusUnit13_11 : Bool;
   //    workpieceStatusUnit14_01 : Bool;
   //    workpieceStatusUnit14_11 : Bool;
   //    workpieceStatusUnit15_01 : Bool;
   //    workpieceStatusUnit15_11 : Bool;
   //    workpieceStatusUnit16_01 : Bool;
   //    workpieceStatusUnit16_11 : Bool;
   //    workpieceStatusUnit17_01 : Bool;
   //    workpieceStatusUnit17_11 : Bool;
   //    workpieceStatusUnit18_01 : Bool;
   //    workpieceStatusUnit18_11 : Bool;
   //    workpieceStatusUnit19_01 : Bool;
   //    workpieceStatusUnit19_11 : Bool;
   //    workpieceStatusUnit20_01 : Bool;
   //    workpieceStatusUnit20_11 : Bool;
   //    workpieceStatusUnit21_01 : Bool;
   //    workpieceStatusUnit21_11 : Bool;
   //    workpieceStatusUnit22_01 : Bool;
   //    workpieceStatusUnit22_11 : Bool;
   //    workpieceStatusUnit23_01 : Bool;
   //    workpieceStatusUnit23_11 : Bool;
   //    workpieceStatusUnit24_01 : Bool;
   //    workpieceStatusUnit24_11 : Bool;
   //    workpieceStatusUnit25_01 : Bool;
   //    workpieceStatusUnit25_11 : Bool;
   //    workpieceStatusUnit26_01 : Bool;
   //    workpieceStatusUnit26_11 : Bool;
   //    workpieceStatusUnit27_01 : Bool;
   //    workpieceStatusUnit27_11 : Bool;
   //    workpieceStatusUnit28_01 : Bool;
   //    workpieceStatusUnit28_11 : Bool;
   //    workpieceStatusUnit29_01 : Bool;
   //    workpieceStatusUnit29_11 : Bool;
   //    workpieceStatusUnit30_01 : Bool;
   //    workpieceStatusUnit30_11 : Bool;
   //    workpieceStatusUnit31_01 : Bool;
   //    workpieceStatusUnit31_11 : Bool;
   //    workpieceStatusUnit32_01 : Bool;
   //    workpieceStatusUnit32_11 : Bool;
   //    workpieceStatusUnit33_01 : Bool;
   //    workpieceStatusUnit33_11 : Bool;
   //    workpieceStatusUnit34_01 : Bool;
   //    workpieceStatusUnit34_11 : Bool;
   //    workpieceStatusUnit35_01 : Bool;
   //    workpieceStatusUnit35_11 : Bool;
   //    workpieceStatusUnit36_01 : Bool;
   //    workpieceStatusUnit36_11 : Bool;
   //    workpieceStatusUnit37_01 : Bool;
   //    workpieceStatusUnit37_11 : Bool;
   //    workpieceStatusUnit38_01 : Bool;
   //    workpieceStatusUnit38_11 : Bool;
   //    workpieceStatusUnit39_01 : Bool;
   //    workpieceStatusUnit39_11 : Bool;
   //    workpieceStatusUnit40_01 : Bool;
   //    workpieceStatusUnit40_11 : Bool;
   //    workpieceCode : Word;
   //    res3092 : Array[3092..3123] of Byte;
   //    identification96Extended : Word;
   //    identification96Extended1 : Word;
   //    identification96Extended2 : Word;
   //    identification96Extended3 : Word;
   //    identification96Extended4 : Word;
   //    identification96Extended5 : Word;
   //    res51 : Array[3136..3144] of Byte;
   //    mach96ExtendedAlarm1 : Word;
   //    toolGroup : Array[1..96] of Struct
   //       toollifeActValue : DWord;
   //       prealarmLinit : DWord;
   //       extendedAlarm : DWord;
   //       alarmLinit : DWord;
   //    END_STRUCT;
   //    workpieceMonitoring : Array[1..112] of Struct
   //       setpoint : DInt;
   //       setpoint2 : DInt;
   //       actualValue : DInt;
   //    END_STRUCT;
   // END_VAR
BEGIN
END_DATA_BLOCK
